	pinPVGTemp.stError:= lib500.IO_PVG_SetOutput(
								pvg_channel:= pinPVGTemp.byChannel,
								output_value:= pinPVGTemp.wValue
							);		
							
	pinPVGTemp.stGetVoltageError := lib500.IO_PVG_GetVoltage(
								pvg_channel:= pinPVGTemp.byChannel,
								voltage:= ADR(pinPVGTemp.uiReadVoltage),
								fresh:= ADR(pinPVGTemp.bVoltageFresh)
							);		
		
	IF pinPVGTemp.stError = lib500_types.IO_ERRORTYPE.IO_E_FET_PROT_REENABLE THEN
		lib500.IO_PVG_ResetProtection(pvg_channel:= pinPVGTemp.byChannel, ADR(pinPowerTemp.byResetCount));
	END_IF
		
	IF (pinPVGTemp.stError <> lib500_types.IO_ERRORTYPE.IO_E_OK AND pinPVGTemp.stError <> lib500_types.IO_ERRORTYPE.IO_E_NO_DIAG) THEN 
		setOutputs:= FALSE; 
		outputPinError:= pinPVGTemp.stError;
	END_IF		
	IF (pinPVGTemp.stGetVoltageError <> lib500_types.IO_ERRORTYPE.IO_E_OK AND pinPVGTemp.stError <> lib500_types.IO_ERRORTYPE.IO_E_NO_DIAG) THEN 
		setOutputs:= FALSE; 
		outputPinError:= pinPVGTemp.stGetVoltageError;
	END_IF
	
	paAllPVGOutputs[iPVGIterator]^:= pinPVGTemp;	
END_FOR
END_METHOD

METHOD PUBLIC mngErrors
VAR_INPUT
END_VAR
ERR.xInputPins:= (inputPinError <> lib500_types.IO_ERRORTYPE.IO_E_OK );
ERR.xOutputPins:= (outputPinError <> lib500_types.IO_ERRORTYPE.IO_E_OK );
ERR.xInitializePins:= (initializePinError <> lib500_types.IO_ERRORTYPE.IO_E_OK );
END_METHOD

END_PROGRAM

// Device/Application/Program logic/UI_PRG
PROGRAM UI_PRG
VAR
	blinker_100ms: BLINK;
	blinker_500ms: BLINK;
END_VAR

blinker_100ms(ENABLE:= TRUE, TIMELOW:= T#100MS, TIMEHIGH:= T#100MS, OUT=> ui.xBlinker_100ms);
blinker_500ms(ENABLE:= TRUE, TIMELOW:= T#500MS, TIMEHIGH:= T#500MS, OUT=> ui.xBlinker_500ms);

END_PROGRAM

// Device/Application/Program logic/mngCanbusStatus
PROGRAM mngCanbusStatus
VAR
	iCanIterator: INT;
	bTmpCanToReinit: BOOL;
	tmpCanStatus: CanHandleStatus;
	handleCloseError: CL2.ERROR;
END_VAR

FOR iCanIterator:= 0 TO fieldbus.iCanbusCount-1 BY 1 DO	
	IF (fieldbus.can[iCanIterator].stChannel.bInitialized) AND fieldbus.can[iCanIterator].bActive THEN
		
		tmpCanStatus:= checkCanBusStatus(
							hDriver:= fieldbus.can[iCanIterator].stChannel.driver, 
							bDriverToReinitialize=> bTmpCanToReinit
						);
						
		IF bTmpCanToReinit THEN
			handleCloseError:= CL2.DriverClose(hDriver:= fieldbus.can[iCanIterator].stChannel.driver);
			fieldbus.can[iCanIterator].stChannel.driver:= CL2.CAA.gc_hINVALID;
			fieldbus.can[iCanIterator].stChannel.bInitialized:= FALSE;
			
			fieldbus.bCanbusInitialized:= initializeCanbus();
			J1939_PRG.xInitialized:= FALSE; // triggers receive mask recreation
		END_IF
		
	END_IF		
END_FOR

METHOD PUBLIC checkCanBusStatus: CanHandleStatus;
VAR_INPUT
	hDriver: CL2.CAA.HANDLE;
END_VAR

VAR_OUTPUT
	bDriverToReinitialize: BOOL;
END_VAR

VAR
	handlerStatus: CanHandleStatus;
	uidFreeMessagesInPoll: UDINT;
	uidMessagesInElabQueue: UDINT;
END_VAR
uidFreeMessagesInPoll:= CL2.GetReceivePoolSize(hDriver, 0);
uidMessagesInElabQueue:= CL2.GetReceiveQueueLength(hDriver, 0);
IF uidFreeMessagesInPoll < CONST.CANBUS_MIN_FREE_POLL OR uidMessagesInElabQueue > CONST.CANBUS_MAX_RX_QUEUE THEN
	ERR.xCanbusHeavy:= TRUE;
	bDriverToReinitialize:= TRUE;
END_IF

handlerStatus.uidFreeMessagesInPoll:= uidFreeMessagesInPoll;
handlerStatus.uidMessagesInElabQueue:= uidMessagesInElabQueue;

checkCanBusStatus:= handlerStatus;
END_METHOD

END_PROGRAM

// Device/Application/Program logic/initializeCanbus
FUNCTION initializeCanbus : BOOL
VAR_INPUT
END_VAR

VAR
	iCanIterator: INT;
	bTempCanbusInitialized: BOOL:= FALSE;
END_VAR

(* initialization of all canbus channels activated by usercode (bActive flag) *)
FOR iCanIterator:= 0 TO fieldbus.iCanbusCount-1 BY 1 DO	
	IF (NOT fieldbus.can[iCanIterator].stChannel.bInitialized) AND fieldbus.can[iCanIterator].bActive THEN			
		fieldbus.can[iCanIterator].stChannel.usiChannel:= INT_TO_USINT(iCanIterator);
		fieldbus.can[iCanIterator].stChannel.uiBaudrateKbps:= fieldbus.uiaCanBaudrates[iCanIterator];
		initializeCanHandle(stCanBus:=fieldbus.can[iCanIterator]);								
	END_IF		
END_FOR

(* check if all activated channels are correctly initialized *)
bTempCanbusInitialized:= TRUE;	
FOR iCanIterator:= 0 TO fieldbus.iCanbusCount-1 BY 1 DO
	IF(fieldbus.can[iCanIterator].bActive AND (NOT fieldbus.can[iCanIterator].stChannel.bInitialized)) THEN
		bTempCanbusInitialized:= FALSE;
		EXIT;
	END_IF
END_FOR

initializeCanbus:= bTempCanbusInitialized;

END_FUNCTION

// Device/Application/Modules/Canbus/Functions/initializeCanHandle
// This PRG contains non safety-related code.
// The following attribute is autogenerated. Do not remove.
{attribute 'location':='16#800'}
PROGRAM initializeCanHandle
VAR_IN_OUT
	stCanBus: canBus;
END_VAR

IF(stCanBus.stChannel.driver = CL2.CAA.gc_hINVALID) THEN
	stCanBus.stChannel.driver := CL2.DriverOpenH(
		usiNetId := stCanBus.stChannel.usiChannel, 
		uiBaudrate := stCanBus.stChannel.uiBaudrateKbps, 
		xSupport29Bits := TRUE, 
		ctMessages := 50, 
		peError := ADR(stCanBus.stChannel.initializeError)
	);		
	IF stCanBus.stChannel.driver <> CL2.CAA.gc_hINVALID  THEN
		stCanBus.stChannel.bInitialized := TRUE;
	END_IF
END_IF

END_PROGRAM

// Device/Application/Modules/J1939/J1939_PRG
PROGRAM J1939_PRG
VAR_INPUT	
	canbus: canBus;
	xInitialized: BOOL:= FALSE;
END_VAR
VAR CONSTANT
	PGN_ONREQ_COUNT: UINT:= 4;
END_VAR
VAR	
	uiLifetimeMs: UINT;
	stJ1939ReceiveMask: canReceiveMask;
	uiPGNRequestSendTimerMs: UINT:= 0;
	byPGNRequestCursor: BYTE:= 0;
	uiaPGNRequestIDs: ARRAY[0..PGN_ONREQ_COUNT-1] OF UINT:= [
		//16#C100,
		16#FEE9,
		16#FEDC,
		//16#FEEB,
		//16#FEDA,
		//16#FEC0,
		16#FEE5,
		16#FDC6
	];
END_VAR

IF NOT xInitialized THEN
	xInitialized:= initReceiveMasks();
ELSE
	receiveMessage();
	IF J1939.xSendPGNRequest THEN sendPGNRequests(); END_IF
END_IF

mngEngineStatus();

Utils.decrementUINT(uiLifetimeMs, 10);

METHOD PRIVATE initReceiveMasks: BOOL;
VAR
	xRet: BOOL:= FALSE;
END_VAR
IF canbus.bActive AND canbus.stChannel.bInitialized THEN
	xRet:= TRUE;
	
	registerReceiveMask(stCanBus:=canbus, udiId:= 16#FFFFFF00, receiveMask:= stJ1939ReceiveMask, udiCobIdMask:= 16#000000FF);
	IF NOT stJ1939ReceiveMask.bInitialized THEN xRet:= FALSE; END_IF

END_IF

initReceiveMasks:= xRet;
END_METHOD

METHOD PRIVATE receiveMessage
VAR CONSTANT
	MAX_RCV_LOOP: UINT:= 100;
END_VAR
VAR
	uiReceivedMsgs: UINT:= 0;
	hMsg: DWORD;
	ctMsgLeft: CL2.CAA.COUNT;
	faulta: CL2.CAA.ERROR;
	udiId: UDINT;
	usiaData: ARRAY[0..7] OF USINT;
END_VAR
REPEAT
	//receive a message from hReceiver
	hMsg := CL2.Read(hReceiverId := stJ1939ReceiveMask.stCAAMask, pctMsgLeft := ADR(ctMsgLeft), peError := ADR(faulta));
	IF hMsg <> 0 THEN
		uiLifetimeMs:= 3000;
		udiId:= CL2.GetMessageId(hMsg, 0);
		usiaData:= CL2.GetMessageDataPointer(hMsg, 0)^;
		
		parseMessage(
			udiMsgId:= udiId, 
			usiData:= usiaData
		);
		
		IF J1939.xRedirectMessages THEN
			redirectToDisplay(
				udiMsgId:= udiId, 
				usiData:= usiaData
			);
		END_IF
		
		CL2.FreeMessage(hMsg); //release message
		hMsg := 0; //to avoid using an already released message
		
	END_IF
UNTIL (ctMsgLeft = 0 OR uiReceivedMsgs > MAX_RCV_LOOP)
END_REPEAT
END_METHOD

METHOD PRIVATE parseMessage
VAR_INPUT	
	udiMsgId: UDINT;
	usiData: ARRAY [0..7] OF USINT;
END_VAR
VAR
	uiPGN: UINT;
	rTmp: REAL;
END_VAR
uiPGN:= UDINT_TO_UINT(SHR(udiMsgId AND 16#00FFFF00, 8));

CASE uiPGN OF
	16#C100:
		J1939.uiMinutesRunWhileMILAct:= Utils.bytesToUInt16(usiData[5], usiData[4]);
		
	16#F004:
		J1939.iTorquePercent:= USINT_TO_INT(usiData[2]) -125;
		J1939.uiEngineSpeedRpm:= REAL_TO_UINT(Utils.bytesToUReal16(usiData[4], usiData[3]) * 0.125);
		
	16#FEE9:
		J1939.lrEngineTotalFuelUsedLiters:= (UDINT_TO_REAL(Utils.bytesToUDInt32(usiData[4], usiData[5], usiData[6], usiData[7])) * 0.5);
		
	16#FEF2:
		J1939.rEngineFuelRateLph:= Utils.bytesToUReal16(usiData[1], usiData[0]) * 0.05;
		
	16#FEF5:
		J1939.byBarometricPressureKPa:= REAL_TO_BYTE(USINT_TO_REAL(usiData[0]) * 0.5);	
		J1939.iAmbientAirTemperatureDegC:= REAL_TO_INT((Utils.bytesToUReal16(usiData[4], usiData[3]) * 0.03125)-273);	
		J1939.iEngineIntakeAirTemperatureDegC:= USINT_TO_INT(usiData[5]) - 40;	
		
	16#FEEF:
		J1939.uiOilPressureKPa:= usiData[3] * 4;	
		J1939.byCoolantLevelPerc:= REAL_TO_BYTE(BYTE_TO_REAL(usiData[7]) * 0.4);	
		
	16#FEEE:
		J1939.iEngineCoolantTempDegC:= USINT_TO_INT(usiData[0]) - 40;	
		J1939.iEngineFuelTempDegC:= USINT_TO_INT(usiData[1]) - 40;	
		
	16#FDB4:
		J1939.iAftertreatmentDPFIntakeGasTempDegC:= (REAL_TO_INT(Utils.bytesToUReal16(usiData[3], usiData[2]) * 0.03125))-273;	
			
	16#FE56:
		;// non chiaro
		
	16#FEF7:
		rTmp:= Utils.bytesToUReal16(usiData[5], usiData[4]);
		IF rTmp = 16#FFFF THEN rTmp:= 0; END_IF
		J1939.rBatteryPotentialV:= rTmp * 0.05;	
		
	16#FDC6:
		J1939.byEngineStartEnable:= usiData[0] AND 16#03;	
		
	16#FEDC:
		J1939.rEngineTotalIdleHours:= (UDINT_TO_REAL(Utils.bytesToUDInt32(usiData[4],usiData[5],usiData[6],usiData[7])) * 0.05);	
		
	16#FC31:
		J1939.byAftertreatmentEngineSpeedIncreaseRequest:= SHR(usiData[0], 4) AND 16#03;	

	16#FEE3:
		;// non chiaro
		
	16#FEEB:
		;// non chiaro

	16#FEE4:
		J1939.byEngineWaitToStartLamp:= usiData[3] AND 16#03;	
		J1939.byEngineIdleShutdownStatus:= usiData[0] AND 16#03;	
		J1939.byEngineIdleShutdownAlert:= SHR(usiData[0], 2) AND 16#03;	
		
	16#FEDA:
		;// non chiaro

	16#FEC0:
		J1939.byServiceComponentId1:= usiData[0];
		J1939.byServiceComponentId2:= usiData[3];
		J1939.byServiceComponentId3:= usiData[5];	
		J1939.iServiceDelayHours:= UINT_TO_INT(Utils.bytesToUInt16(usiData[7],usiData[6])) - 32127;	

	16#FEE5:
		J1939.rEngineTotalOperationHours:= (UDINT_TO_REAL(Utils.bytesToUDInt32(usiData[0],usiData[1],usiData[2],usiData[3])) * 0.05);	
	
	16#FD7C:
		J1939.byDPFFilterLamp:= usiData[0] AND 16#07;	
		J1939.byAftertreatmentDPFActiveRegeneration:= SHR(usiData[1], 2) AND 16#03;	
		J1939.byAftertreatmentDPFFilterStatus:= SHR(usiData[1], 4) AND 16#07;	
		J1939.byDPFActiveRegenerationInhibitedDueSwitch:= SHR(usiData[2], 2) AND 16#03;	
		J1939.byDPFActiveRegenerationInhibitedDueTmpSysLock:= usiData[5] AND 16#03;	
		J1939.byDPFActiveRegenerationInhibitedDuePermSysLock:= SHR(usiData[5], 2) AND 16#03;	
		
	16#FECA:
		J1939.byWarningIndicator:= SHR(usiData[0], 2) AND 16#03;	
		J1939.byWarningIndicatorFlash:= SHR(usiData[1], 2) AND 16#03;
		J1939.byShutdownIndicator:= SHR(usiData[0], 4) AND 16#03;
		J1939.byEngineProtectIndicator:= SHR(usiData[0], 0) AND 16#03;
		J1939.byEngineProtectIndicatorFlash:= SHR(usiData[1], 0) AND 16#03;
		J1939.byEmissionSystemMalfunctionIndicator:= SHR(usiData[0], 6) AND 16#03;
		J1939.byEmissionSystemMalfunctionIndicatorFlash:= SHR(usiData[1], 6) AND 16#03;

		J1939.DM1_SPN:= usiData[2];
		J1939.DM1_SPN:= J1939.DM1_SPN OR SHL(BYTE_TO_ULINT(usiData[3]), 8);
		J1939.DM1_SPN:= J1939.DM1_SPN OR SHL(BYTE_TO_ULINT(usiData[4] AND 16#E0), 16);
		IF J1939.DM1_SPN = 16#7FFFF THEN J1939.DM1_SPN:= 0; END_IF
		J1939.DM1_FMI:= usiData[4] AND 16#1F;
		IF J1939.DM1_FMI = 16#1F THEN J1939.DM1_FMI:= 0; END_IF
		J1939.DM1_OC:= usiData[5] AND 16#7F;
		IF J1939.DM1_OC = 16#7F THEN J1939.DM1_OC:= 0; END_IF
		
	16#FD0C: // NON C'E'
		// J1939.xLowOilPressure:= (SHR(usiData[1], 4) AND 16#03) = 1;	
	
END_CASE
END_METHOD

METHOD PRIVATE sendPGNRequests
VAR
	i: INT;
	msg: canMessage;
END_VAR
Utils.decrementUINT(uiPGNRequestSendTimerMs, 10);
IF uiPGNRequestSendTimerMs > 0 THEN RETURN; END_IF
uiPGNRequestSendTimerMs:= 100;

msg.bExtended:= TRUE;
msg.byLength:= 3;
msg.udiId:= 16#18EAFF00;
msg.udiId:= msg.udiId OR J1939.byECUNodeId;
msg.byaData[0]:= UINT_TO_BYTE(SHR(uiaPGNRequestIDs[byPGNRequestCursor], 0) AND 16#FF);
msg.byaData[1]:= UINT_TO_BYTE(SHR(uiaPGNRequestIDs[byPGNRequestCursor], 8) AND 16#FF);
msg.byaData[2]:= 0;

byPGNRequestCursor:= byPGNRequestCursor+1;
IF byPGNRequestCursor >= PGN_ONREQ_COUNT THEN 
	byPGNRequestCursor:= 0;
END_IF

sendMessage(stCanBus:= canbus, stMessageToSend:= msg);
END_METHOD

METHOD PUBLIC mngEngineStatus
VAR_INPUT
END_VAR
J1939.xEngineOnline:= uiLifetimeMs > 0;

J1939.xEngineRunning:= J1939.xEngineOnline AND (J1939.uiEngineSpeedRpm > 300);
J1939.xEngineDPFRegenActive:= J1939.xEngineOnline AND (J1939.byAftertreatmentDPFActiveRegeneration = 1);
J1939.xEngineDPFRegenRequest:= J1939.xEngineOnline AND (J1939.byAftertreatmentDPFActiveRegeneration = 2);

J1939.xLowOilPressure:= (J1939.uiOilPressureKPa < 90);

J1939.xEngineLamp:= (
		J1939.byWarningIndicator = 1 OR	
		J1939.byWarningIndicatorFlash = 1 OR	
		J1939.byEngineProtectIndicator = 1 OR	
		J1939.byEngineProtectIndicatorFlash = 1 OR	
		J1939.byEmissionSystemMalfunctionIndicator = 1 OR	
		J1939.byEmissionSystemMalfunctionIndicatorFlash = 1
);	

J1939.xEngineLampRed:= (
	J1939.byShutdownIndicator = 1
);
END_METHOD

METHOD PRIVATE redirectToDisplay
VAR_INPUT	
	udiMsgId: UDINT;
	usiData: ARRAY [0..7] OF USINT;
END_VAR
VAR
	msg: canMessage;
	i: INT;
END_VAR
msg.udiId:= udiMsgId;
msg.byLength:= 8;
msg.bExtended:= TRUE;
FOR i:= 0 TO 7 DO
	msg.byaData[i]:= USINT_TO_BYTE(usiData[i]);
END_FOR

sendMessage(stCanBus:= fieldbus.can[2], stMessageToSend:= msg);
END_METHOD

END_PROGRAM

// Device/Application/Program logic/Tasks/MachineLogic_PRG
PROGRAM MachineLogic_PRG
VAR CONSTANT
	dwDuty_half: UINT:= 16#4FFF;
	dwDuty_on: UINT:= 16#FFFF;
	dwDuty_off: UINT:= 16#0000;
END_VAR
VAR
	uiSeatTimerMs: UINT;
	
	xKeyInput: BOOL;
	xGearEngaged: BOOL;
	xSlowGearEngaged: BOOL;
	xTractionMoving: BOOL;
	xInchingConditionsMet: BOOL;
	
	xForwardGear: BOOL;
	xReverseGear: BOOL;
	
	xForwardInching: BOOL;
	xReverseInching: BOOL;
	
	xOilOvertemperature: BOOL;
	
	udiInchingActiveTimerMs: UDINT;
	uiInchingBrakeTimerMs: UINT;
	
	uiIncorrectStartReload: UINT:= 1000;
	uiIncorrectStartTimer: UINT:= uiIncorrectStartReload;
	
	xMachineAutodetectInit: BOOL:= FALSE;
	
	xParkingBrakeButtonStatus: BOOL;
	uiPBrakeButtonAntibounceTimerMs: UINT;
	
	dwEncoderValueOld_p151: DWORD;
	uiEncoderReadFreshTimerMs_p151: UINT;
	xEncoderFresh_p151: BOOL:= FALSE;
	
END_VAR

Cab_C002080();

METHOD Cab_C002080
VAR_INPUT
	
END_VAR
VAR
	temp: word;
END_VAR
 
sysIO.digitalOutput.output_149.bvalue := varOutput.xOutput_1 ;
sysIO.digitalOutput.output_150.bvalue := varOutput.xOutput_2 ;
sysIO.digitalOutput.output_152.bvalue := varOutput.xOutput_3 ;
sysIO.digitalOutput.output_153.bvalue := varOutput.xOutput_4 ;
sysIO.digitalOutput.output_154.bvalue := varOutput.xOutput_5 ;
sysIO.digitalOutput.output_155.bvalue := varOutput.xOutput_6 ;
sysIO.digitalOutput.output_156.bvalue := varOutput.xOutput_7 ;
sysIO.digitalOutput.output_157.bvalue := varOutput.xOutput_8 ;
sysIO.digitalOutput.output_158.bvalue := varOutput.xOutput_9 ;
sysIO.digitalOutput.output_159.bvalue := varOutput.xOutput_10;
sysIO.digitalOutput.output_173.bvalue := varOutput.xOutput_11;
sysIO.digitalOutput.output_174.bvalue := varOutput.xOutput_12;
sysIO.digitalOutput.output_176.bvalue := varOutput.xOutput_13;
sysIO.digitalOutput.output_177.bvalue := varOutput.xOutput_14;
sysIO.digitalOutput.output_178.bvalue := varOutput.xOutput_15;
sysIO.digitalOutput.output_179.bvalue := varOutput.xOutput_16;
sysIO.digitalOutput.output_180.bvalue := varOutput.xOutput_17;
sysIO.digitalOutput.output_181.bvalue := varOutput.xOutput_18;
sysIO.digitalOutput.output_182.bvalue := varOutput.xOutput_19;
sysIO.digitalOutput.output_183.bvalue := varOutput.xOutput_20;


varInput.xInput_1  := sysIO.digitalInput.input_115.bValue;
varInput.xInput_2  := sysIO.digitalInput.input_116.bValue;
varInput.xInput_3  := sysIO.digitalInput.input_117.bValue;
varInput.xInput_4  := sysIO.digitalInput.input_122.bValue;
varInput.xInput_5  := sysIO.digitalInput.input_123.bValue;
varInput.xInput_6  := sysIO.digitalInput.input_124.bValue;
varInput.xInput_7  := sysIO.digitalInput.input_139.bValue;
varInput.xInput_8  := sysIO.digitalInput.input_140.bValue;
varInput.xInput_9  := sysIO.digitalInput.input_141.bValue;
varInput.xInput_10 := sysIO.digitalInput.input_146.bValue;
varInput.xInput_11 := sysIO.digitalInput.input_147.bValue;
varInput.xInput_12 := sysIO.digitalInput.input_148.bValue;
varInput.xInput_13 := sysIO.digitalInput.input_161.bValue;
varInput.xInput_14 := sysIO.digitalInput.input_164.bValue;
varInput.xInput_15 := sysIO.digitalInput.input_167.bValue;
varInput.xInput_16 := sysIO.digitalInput.input_170.bValue;
varInput.xInput_17 := sysIO.digitalInput.input_185.bValue;
varInput.xInput_18 := sysIO.digitalInput.input_188.bValue;
varInput.xInput_19 := sysIO.digitalInput.input_191.bValue;
varInput.xInput_20 := sysIO.digitalInput.input_194.bValue;
END_METHOD

END_PROGRAM

// Device/Application/Modules/Canbus/Safety interface/Functions/safeSendMessage
PROGRAM safeSendMessage
VAR_IN_OUT
	stCanBus: canBus;
END_VAR
VAR_INPUT
	stMessageToSend: canMessage;
END_VAR
VAR
	iTransMsgPointer: INT:= 0;
END_VAR

FOR iTransMsgPointer:= 0 TO canGVL.iTransmitBufferSize-1 BY 1 DO
	IF(stCanBus.stTransmitBuffer[iTransMsgPointer].udiId = 0) THEN
		stCanBus.stTransmitBuffer[iTransMsgPointer]:= stMessageToSend;
		EXIT;
	END_IF
END_FOR

END_PROGRAM

// Device/Application/Modules/Canbus/Safety interface/Functions/safetyCanbusInterface
PROGRAM safetyCanbusInterface
VAR_INPUT
END_VAR
VAR_OUTPUT
END_VAR
VAR
END_VAR

END_PROGRAM

// Device/Application/Modules/Canbus/Safety interface/Tasks/CAN_PRG_SAFE
PROGRAM CAN_PRG_SAFE
VAR_INPUT
END_VAR
VAR_OUTPUT
END_VAR
VAR
END_VAR

exchangeVariables();

METHOD exchangeVariables
VAR
	iBusCursor: INT;
END_VAR
(* unsafe --> safe *)
IF canEVL.bChannelsHasChanges THEN	
	FOR iBusCursor:= 0 TO canGVL.iBusCount-1 BY 1 DO	
		canGVL.busses[iBusCursor].stChannel:= canGVL.busses[iBusCursor].stChannel;
	END_FOR
	canEVL.bChannelsHasChanges:= FALSE;	
	
ELSIF canEVL.bTransmitBuffersHasChanges THEN	
	FOR iBusCursor:= 0 TO canGVL.iBusCount-1 BY 1 DO	
		canGVL.busses[iBusCursor].stTransmitBuffer:= canGVL.busses[iBusCursor].stTransmitBuffer;
	END_FOR	
	canEVL.bTransmitBuffersHasChanges:= FALSE;
	
ELSIF canEVL.bMasksHasChanges THEN	
	FOR iBusCursor:= 0 TO canGVL.iBusCount-1 BY 1 DO	
		canGVL.busses[iBusCursor].staReceiveMasks:= canGVL.busses[iBusCursor].staReceiveMasks;
	END_FOR	
	canEVL.bMasksHasChanges:= FALSE;
	
END_IF
END_METHOD

END_PROGRAM

// Device/Application/Modules/Canbus/Safety interface/Tasks/CAN_PRG_UNSAFE
// This PRG contains non safety-related code.
// The following attribute is autogenerated. Do not remove.
{attribute 'location':='16#800'}
PROGRAM CAN_PRG_UNSAFE
VAR_INPUT
END_VAR
VAR_OUTPUT
END_VAR
VAR
	iBusCursor: INT:= 0;
	iTransMsgPointer: INT:= 0;
	iReceiveMaskPointer: INT:= 0;
END_VAR

FOR iBusCursor:= 0 TO canGVL.iBusCount-1 BY 1 DO
	
	IF( canGVL.busses[iBusCursor].bActive AND (NOT canGVL.busses[iBusCursor].stChannel.bInitialized) ) THEN
		(* Inizializzazione canali *)
		canEVL.busses[iBusCursor]:= canGVL.busses[iBusCursor];
		initializeCanHandle(stCanBus:=canEVL.busses[iBusCursor]);
		IF canEVL.busses[iBusCursor].stChannel.bInitialized THEN canEVL.bChannelsHasChanges:= TRUE; END_IF;
		
	ELSIF( canGVL.busses[iBusCursor].bActive AND canGVL.busses[iBusCursor].stChannel.bInitialized ) THEN
		
		(* Creazione maschere di ricezione *)
		FOR iReceiveMaskPointer:= 0 TO canGVL.iReceiveMaskCount-1 BY 1 DO
			IF(canGVL.busses[iBusCursor].staReceiveMasks[iReceiveMaskPointer].bActive AND NOT canGVL.busses[iBusCursor].staReceiveMasks[iReceiveMaskPointer].bInitialized) THEN
				registerReceiveMask(stCanBus:= canGVL.busses[iBusCursor], 
									udiId:= canGVL.busses[iBusCursor].staReceiveMasks[iReceiveMaskPointer].udiId,
									receiveMask:= canEVL.busses[iBusCursor].staReceiveMasks[iReceiveMaskPointer]
									); 
				canEVL.bMasksHasChanges:= TRUE;
			END_IF
		END_FOR
		
		(* Invio messaggi *)
		FOR iTransMsgPointer:= 0 TO canGVL.iTransmitBufferSize-1 BY 1 DO
			IF(canGVL.busses[iBusCursor].stTransmitBuffer[iTransMsgPointer].udiId > 0) THEN
				sendMessage(stCanBus:= canGVL.busses[iBusCursor], stMessageToSend:= canGVL.busses[iBusCursor].stTransmitBuffer[iTransMsgPointer]);
				canEVL.busses[iBusCursor].stTransmitBuffer[iTransMsgPointer].udiId:= 0;

				canEVL.bTransmitBuffersHasChanges:= TRUE;
			END_IF
		END_FOR	 
		
	END_IF
	
END_FOR

END_PROGRAM

// Device/Application/Modules/Canbus/Safety interface/Functions/safeRegisterReceiveMask
PROGRAM safeRegisterReceiveMask
VAR_IN_OUT
	stCanBus: canBus;
END_VAR
VAR_INPUT
	udiId: UDINT:= 0;
END_VAR
VAR_OUTPUT
	iMaskCursor: INT:= -1;
END_VAR
VAR
	iReceiveMaskCursor: INT:= 0;
	stNewReceiveMask: canReceiveMask;
END_VAR

FOR iReceiveMaskCursor:= 0 TO canGVL.iReceiveMaskCount-1 BY 1 DO
	IF(NOT stCanBus.staReceiveMasks[iReceiveMaskCursor].bActive) THEN
		stNewReceiveMask.udiId:= udiId;
		stNewReceiveMask.bActive:= TRUE;
		stCanBus.staReceiveMasks[iReceiveMaskCursor]:= stNewReceiveMask;
		iMaskCursor:= iReceiveMaskCursor;
		EXIT;
	END_IF
END_FOR

END_PROGRAM

// Device/Application/Visualization
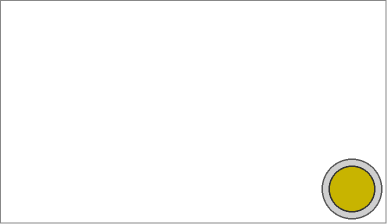
VISUALIZATION Visualization  // 387x224
    Lamp1 (317,154 70x70), invisible if: system.machineModel = 1, style: Lamp-Lamp1-Yellow
END_VISUALIZATION
